(* PLC project Unnamed, 不明 Unnamed 1 *)
(* stored: creationDateTime 2023-01-05T13:54:08, modificationDateTime 2023-01-16T19:29:52 *)

PROGRAM program0
  VAR
    Degital_in_0 AT %IX0.0 : BOOL;
    Degital_in_1 AT %IX0.1 : BOOL;
    Degital_in_2 AT %IX0.2 : BOOL;
    Degital_in_3 AT %IX0.3 : BOOL;
    Degital_in_4 AT %IX0.4 : BOOL;
    Degital_out_0 AT %QX0.0 : BOOL;
    Degital_out_1 AT %QX0.1 : BOOL;
    Degital_out_2 AT %QX0.2 : BOOL;
    Degital_out_3 AT %QX0.3 : BOOL;
    Analog_in_0 AT %IW0 : UINT;
    Analog_in_1 AT %IW1 : UINT;
    Analog_in_2 AT %IW2 : UINT;
    Analog_in_3 AT %IW3 : UINT;
    Analog_in_4 AT %IW4 : UINT;
    Analog_in_5 AT %IW5 : UINT;
    Analog_OUT_0 AT %QW0 : UINT;
    Analog_OUT_1 AT %QW1 : UINT;
    Analog_OUT_2 AT %QW2 : UINT;
  END_VAR

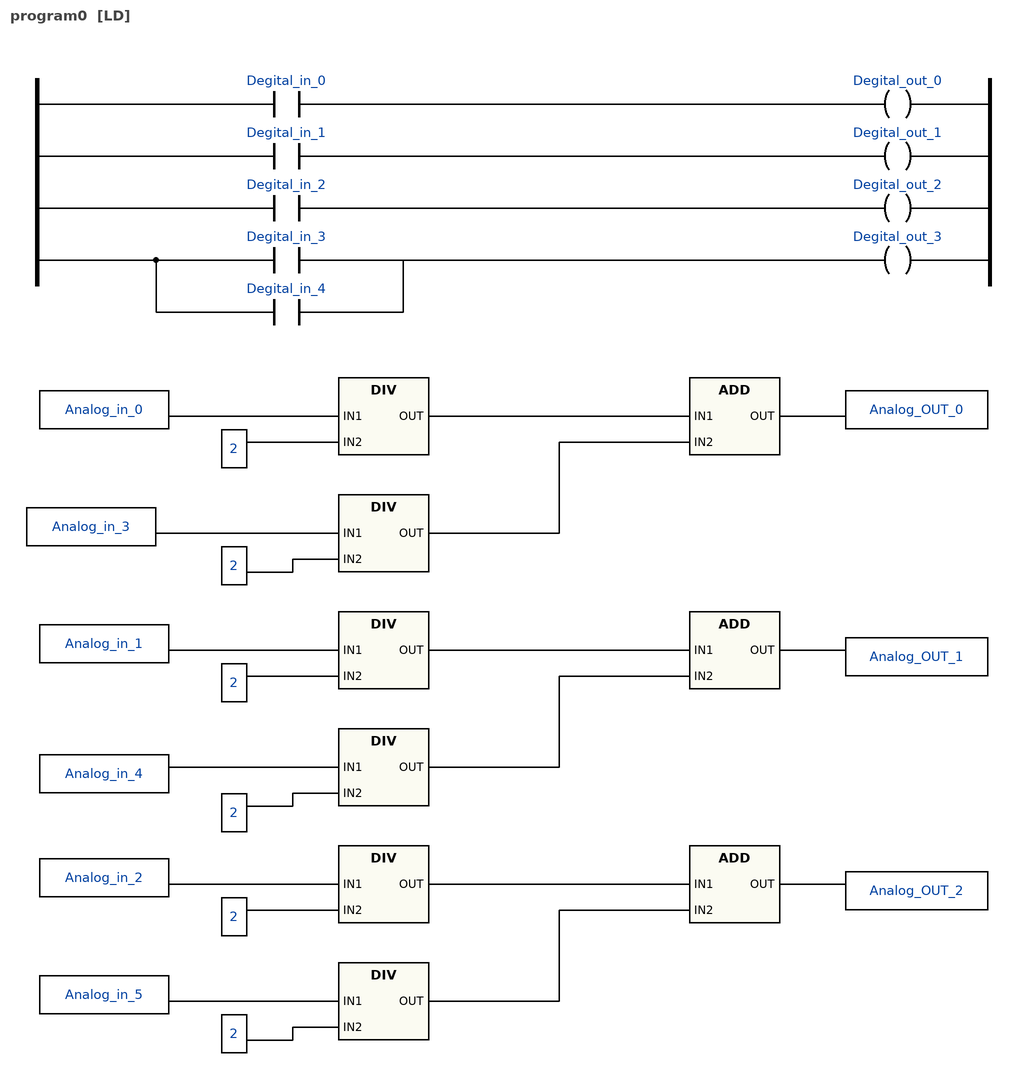
(* LD diagram, written out as Structured Text *)
Degital_out_0 := Degital_in_0;
Degital_out_1 := Degital_in_1;
Degital_out_2 := Degital_in_2;
Degital_out_3 := Degital_in_3 OR Degital_in_4;
Analog_OUT_0 := Analog_in_0 / 2 + Analog_in_3 / 2;
Analog_OUT_1 := Analog_in_1 / 2 + Analog_in_4 / 2;
Analog_OUT_2 := Analog_in_2 / 2 + Analog_in_5 / 2;
END_PROGRAM

CONFIGURATION Config0
  RESOURCE Res0 ON PLC
    TASK task0(INTERVAL := T#20ms, PRIORITY := 0);
    PROGRAM instance0 WITH task0 : program0;
  END_RESOURCE
END_CONFIGURATION
